TYPE CoverPanelParts :
STRUCT
	///NC Axis
	axis: AngularAxis;
	///Relay for the motor
	motorRelay: SimpleRelay;
END_STRUCT
END_TYPE

(* stored: Version 1.1.0.1, ProductVersion 3.1.4019.2
   DUT CoverPanelParts: Id {c5de605e-33b4-45ef-a972-7d3e31b16a60} *)
